# EPICS IOC start-up script: e3-tgt-twds1000_ctrl-plc-01/tgt-twds1000_ctrl-plc-01-loc/iocsh/tgt-twds1000_ctrl-plc-01-test.iocsh
# @field tgt-twds1000_ctrl-plc-01_VERSION
# @runtime YES

# Load plc interface database
dbLoadRecords("tgt-twds1000_ctrl-plc-01-test.db", "MODVERSION=$(tgt-twds1000_ctrl-plc-01_VERSION)")
